// TIA Portal V16 export
// export: Created 2026-06-18T08:15:20.5409663Z, ExportSetting WithDefaults, DisplayName Totally Integrated Automation Portal, DisplayVersion V16 Update 8, DisplayName TIA Portal Version Control Interface, DisplayVersion V16 Update 8, DisplayName TIA Portal Openness, DisplayVersion V16 Update 8, DisplayName SINAMICS Startdrive Advanced, DisplayVersion V16, DisplayName SINAMICS Startdrive G130, G150, S120, S150, SINAMICS MV, S210, DisplayVersion V16, DisplayName SINAMICS Startdrive G110M, G120, G120C, G120D, G120P, DisplayVersion V16, DisplayName STEP 7 Professional, DisplayVersion V16 Update 8, DisplayName STEP 7 Safety, DisplayVersion V16 Update 7, DisplayName WinCC Advanced, DisplayVersion V16 Update 8
Screen "Pipeline_Flow"  800x480, Number=1
  ScreenLayer 
    IOField "IO_FlowInstant" at 170,95 size 160x44  DataFormat=Decimal, FormatPattern=9999999, Mode=InOutput
    IOField "IO_FlowAnimValue" at 170,360 size 120x44  DataFormat=Decimal, FormatPattern=9999999, Mode=InOutput
    IOField "IO_FlowTotal" at 170,155 size 160x44  DataFormat=Decimal, FormatPattern=9999999, Mode=InOutput
    SymbolicIOField "符号 I/O 域_1" at 177,87 size 170x32  CountVisibleItems=3, Mode=InOutput, OnValue=1, TextOff="0", TextOn="1"
    TextField "TXT_Title" at 180,20 size 440x44  Text="管道流量控制"
    Button "BTN_Start" at 420,95 size 130x56  Mode=Text, TextOff="启动", TextOn="启动"
    Button "BTN_Stop" at 580,95 size 130x56  Mode=Text, TextOff="停止", TextOn="停止"
    Circle "LMP_Pump" at 170,240 size 48x48
    Circle "LMP_FlowAnim" at 170,300 size 48x48
